TYPE ST_M2SelectorIO EXTENDS ST_M3DeviceBaseIO:
STRUCT


	
END_STRUCT
END_TYPE

(* stored: Version 1.1.0.1, ProductVersion 3.1.4022.18
   DUT ST_M2SelectorIO: Id {8847cae4-58e8-4ecd-b246-7e3fca7dfce8} *)
